{attribute 'GeneratedUsingTerminal: AX8206-0100-0101-0101'}
{attribute addProperty BoxType "AX8206-0100-0101-0101"}
{attribute addProperty Id "DeviceDevice_6E2575772Device_SafetyDevice_Safety_C21945A160Ch_ACh_A_1FF86D8522Ch_BCh_B_5E084BAA22WcStateAT %I*WcState_B516A2644InfoDataAT %I*InfoData_FD1CC0AA12"}
{attribute addProperty CRC "3021183848"}
{attribute addProperty Size "122"}
TYPE AX8206_B4139B68 EXTENDS EtcSlaveTerminalBase_947E5A46 :
STRUCT
	{attribute addProperty Name "Device"}
	Device : Device_6E257577;
	{attribute addProperty Name "Device_Safety"}
	Device_Safety : Device_Safety_C21945A1;
	{attribute addProperty Name "Ch_A"}
	Ch_A : Ch_A_1FF86D85;
	{attribute addProperty Name "Ch_B"}
	Ch_B : Ch_B_5E084BAA;
	{attribute addProperty Name "WcState"}
	WcState : WcState_B516A264;
	{attribute addProperty Name "InfoData"}
	InfoData : InfoData_FD1CC0AA;
END_STRUCT
END_TYPE

(* stored: Version 1.2.0.0, ProductVersion 3.1.4024.9
   DUT AX8206_B4139B68: Id {fa12c8f4-068c-4601-851c-89c45b872c59} *)
